FUNCTION_BLOCK registerLogic (* Basic Function Block Type *)
  (* Standard: 61499-2 *)
  (* Version 0.0, 8/1/2013, herrric, nxtControl GmbH, Template *)
  PACKAGE Loytec.Communication;
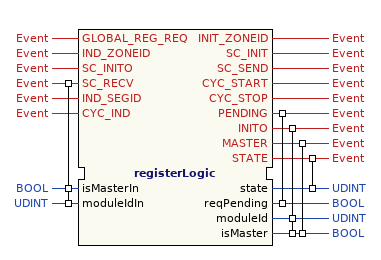
  EVENT_INPUT
    GLOBAL_REG_REQ; (* Initialization Request *)
    IND_ZONEID;
    SC_INITO;
    SC_RECV WITH isMasterIn, moduleIdIn;
    IND_SEGID;
    CYC_IND;
  END_EVENT
  EVENT_OUTPUT
    INIT_ZONEID; (* Initialization Confirm *)
    SC_INIT;
    SC_SEND;
    CYC_START;
    CYC_STOP;
    PENDING WITH reqPending;
    INITO WITH moduleId, isMaster;
    MASTER WITH isMaster;
    STATE WITH state;
  END_EVENT
  VAR_INPUT
    isMasterIn : BOOL;
    moduleIdIn : UDINT;
  END_VAR
  VAR_OUTPUT
    state : UDINT;
    reqPending : BOOL;
    moduleId : UDINT;
    isMaster : BOOL;
  END_VAR
  VAR
    zoneIdAvailable : BOOL := FALSE;
  END_VAR
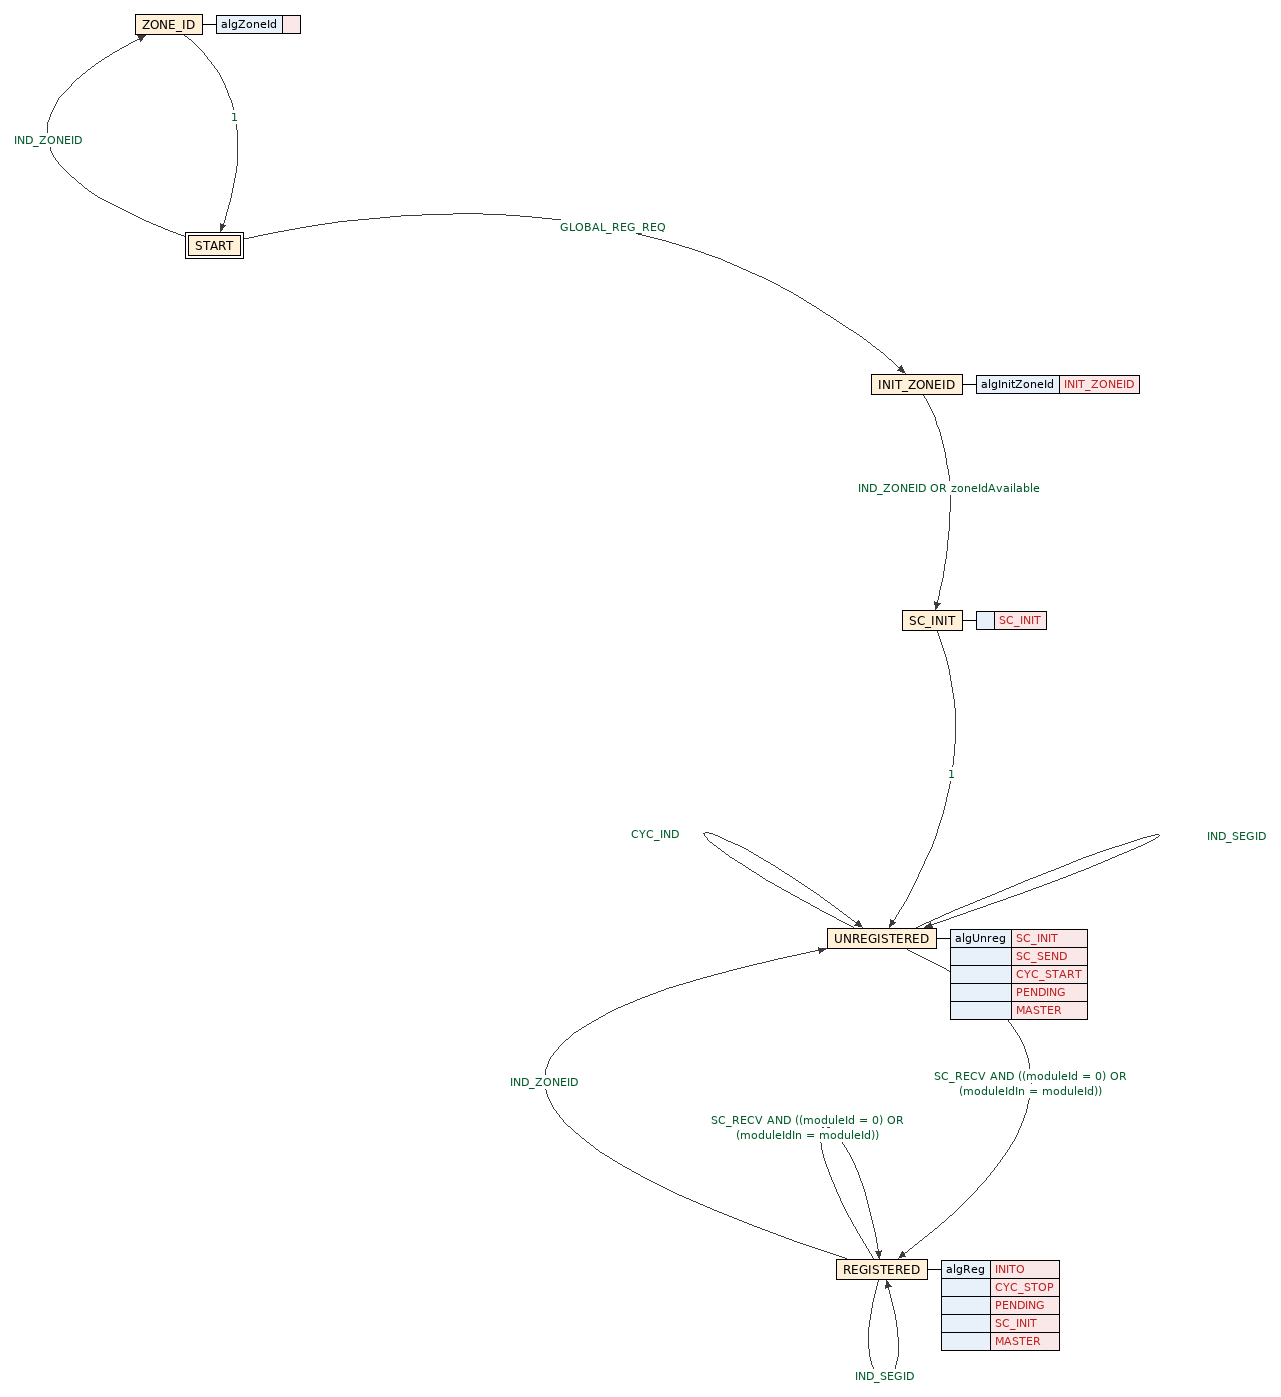
  EC_STATES
    START; (* Initial State *)
    INIT_ZONEID : algInitZoneId -> INIT_ZONEID;
    UNREGISTERED : algUnreg -> SC_INIT, -> SC_SEND, -> CYC_START, -> PENDING, -> MASTER;
    REGISTERED : algReg -> INITO, -> CYC_STOP, -> PENDING, -> SC_INIT, -> MASTER;
    SC_INIT : -> SC_INIT;
    ZONE_ID : algZoneId;
  END_STATES
  EC_TRANSITIONS
    START TO INIT_ZONEID := GLOBAL_REG_REQ;
    INIT_ZONEID TO SC_INIT := IND_ZONEID OR zoneIdAvailable;
    UNREGISTERED TO REGISTERED := SC_RECV AND ((moduleId = 0) OR (moduleIdIn = moduleId));
    REGISTERED TO UNREGISTERED := IND_ZONEID;
    REGISTERED TO REGISTERED := IND_SEGID;
    UNREGISTERED TO UNREGISTERED := IND_SEGID;
    UNREGISTERED TO UNREGISTERED := CYC_IND;
    START TO ZONE_ID := IND_ZONEID;
    ZONE_ID TO START := 1;
    SC_INIT TO UNREGISTERED := 1;
    REGISTERED TO REGISTERED := SC_RECV AND ((moduleId = 0) OR (moduleIdIn = moduleId));
  END_TRANSITIONS
  ALGORITHM algUnreg IN ST:
state := 1;
SC_INIT := IND_SEGID;
reqPending := TRUE;

IF isMaster = TRUE THEN
	isMaster := FALSE;
ELSE
	MASTER := FALSE;
END_IF;
  END_ALGORITHM
  ALGORITHM algReg IN ST:
state := 2;
reqPending := FALSE;

IF moduleId = 0 OR moduleId = moduleIdIn THEN
	moduleId := moduleIdIn;
	IF isMaster <> isMasterIn THEN
		isMaster := isMasterIn;
	ELSE
		MASTER := FALSE;
	END_IF;
ELSE
	MASTER := FALSE;
	INITO := FALSE;
END_IF;

SC_RECV := FALSE;
  END_ALGORITHM
  ALGORITHM algZoneId IN ST:
zoneIdAvailable := TRUE;
  END_ALGORITHM
  ALGORITHM algInitZoneId IN ST:
IF zoneIdAvailable THEN
	INIT_ZONEID := FALSE;
END_IF;
  END_ALGORITHM
END_FUNCTION_BLOCK
